{attribute 'GeneratedUsingTerminal: BK1120-0000-0000'}
{attribute addProperty BoxType "BK1120-0000-0000"}
{attribute addProperty Id "Term_374_KL1002KL1002_BB38DA8F0"}
{attribute addProperty CRC "543057241"}
{attribute addProperty Size "0"}
TYPE A_0001_BK1120_0000_0000_205E6559 EXTENDS BK1120_DB80BFFC :
STRUCT
	{attribute addProperty Name "Term_374_KL1002"}
	Term_374_KL1002 : KL1002_BB38DA8F;
END_STRUCT
END_TYPE

(* stored: Version 1.2.0.0, ProductVersion 3.1.4024.9
   DUT A_0001_BK1120_0000_0000_205E6559: Id {16074ed1-cf34-4d4f-bc42-0d6a5b0783db} *)
